Fanuc KAREL source: ka00132.KL

PROGRAM KA00132
%STACKSIZE=65535
%PRIORITY=65535
%NOLOCKGROUP
-- UNRESOLVED DECLARATIONS (source type spelling not recovered)
-- SRC : ARRAY[2] OF TYPE_0x0018 (type_u16=0x2018)
-- DST : ARRAY[2] OF TYPE_0x0017 (type_u16=0x2017)
BEGIN
SRC[1]=2
-- UNRESOLVED_PC line 8 opcodes [22 9D 33 B1 22 9D 33 B4] marker_code=19
END KA00132
